PROGRAM LogProgram
VAR_INPUT
	State: INT :=0;
	NewState: INT := 0;

END_VAR

VAR
	bStart: BOOL;		// Start the sequence
END_VAR

///////////////////////////// For logging of datas /////////////////////////////
IF bLog THEN
	bStart := TRUE;
	
ELSE 
	bStart := FALSE;
END_IF

CASE State OF

	0:	
		tLogTime.IN 		:= FALSE;
		uiElapsedTime		:= 0;
		usiImageLog			:= 0;
		usiStickoutCutLog	:= 0;
		usiRetryLog			:= 0;
		usiImageRetry		:= 0;
		bLogSucces			:= 0;
		IF bStart THEN
			bStart := FALSE;
			tLogTime.IN := TRUE;
			NewState := 10;
		END_IF
		
	10:		// Check if all states are in state 0	-	This means that the sequence has finished
		IF (Tools.State = 0) AND (Control.State = 0) THEN
			bLog := FALSE;
			uiElapsedTime := TO_UINT(tLogTime.ET);
			NewState := 20;
		END_IF 
		
	20:
		P_SqlInsertLog.bInsert := TRUE;
		IF P_SqlInsertLog.bDone THEN
			P_SqlInsertLog.bInsert := FALSE;
			NewState := 0;
		END_IF

END_CASE


(*
	bLog:				BOOL;		// For logging of data
	tLogTime:			TON;		// Time for one sequence
	usiImageLog:		USINT;		// Counting number of images taken in a sequence
	usiStickoutCutLog:	USINT;		// For counting number of stick-outs
	bLogSucces:			BOOL;		// TRUE if success	-	FALSE if not
*)

///////////////////////////// Timers /////////////////////////////
tLogTime (PT := T#5M);

END_PROGRAM

(* stored: Version 1.1.0.1, ProductVersion 3.1.4024.4
   POU LogProgram: Id {c551ccbb-dc84-4d9c-829d-76540082eb74}, SpecialFunc None *)
